// LS Electric XG5000 project: 7k_pwm_20190129_HMI타이밍변경
// PLC NewPLC
// module base 0 slot 0: 입출력 모듈:XBM-DN/DP32H2 (DC 24V입력/TR 출력, 32점)
// module base 0 slot 1: 내장위치결정:XBF-PO02E (오픈컬렉터형, 2축)

PROGRAM 7k_pwm (task: 스캔 프로그램)

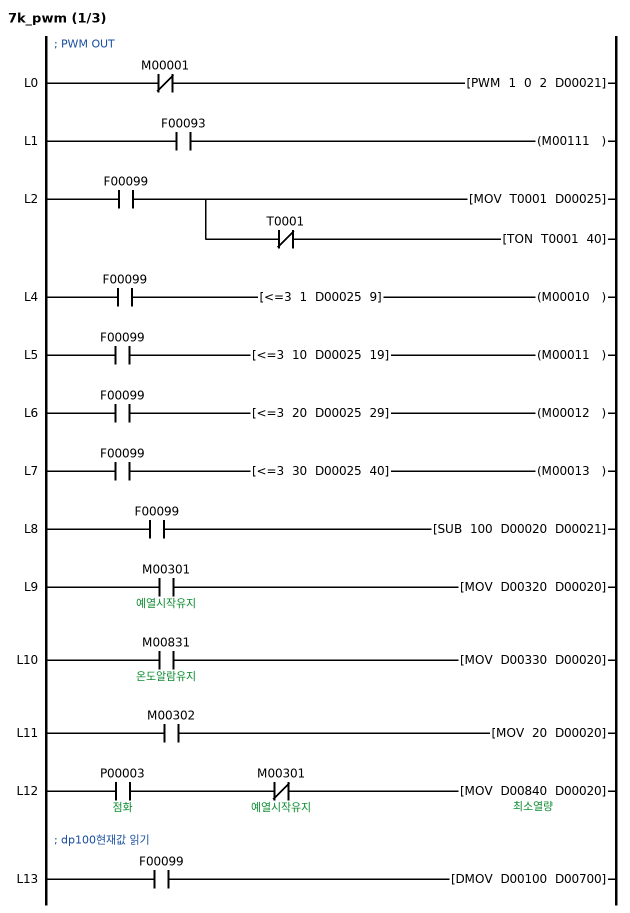
; L0
LOAD NOT  M00001
PWM       1 0 2 D00021
// output comment: PWM OUT
; L1
LOAD      F00093
OUT       M00111
; L2
LOAD      F00099
MOV       T0001 D00025
AND NOT   T0001
TON       T0001 40
; L4
LOAD      F00099
AND<=3    1 D00025 9
OUT       M00010
; L5
LOAD      F00099
AND<=3    10 D00025 19
OUT       M00011
; L6
LOAD      F00099
AND<=3    20 D00025 29
OUT       M00012
; L7
LOAD      F00099
AND<=3    30 D00025 40
OUT       M00013
; L8
LOAD      F00099
SUB       100 D00020 D00021
; L9
LOAD      M00301	// 예열시작유지
MOV       D00320 D00020
; L10
LOAD      M00831	// 온도알람유지
MOV       D00330 D00020
; L11
LOAD      M00302
MOV       20 D00020
; L12
LOAD      P00003	// 점화
AND NOT   M00301	// 예열시작유지
MOV       D00840 D00020	// 최소열량
; L13
LOAD      F00099
DMOV      D00100 D00700
// output comment: dp100현재값 읽기

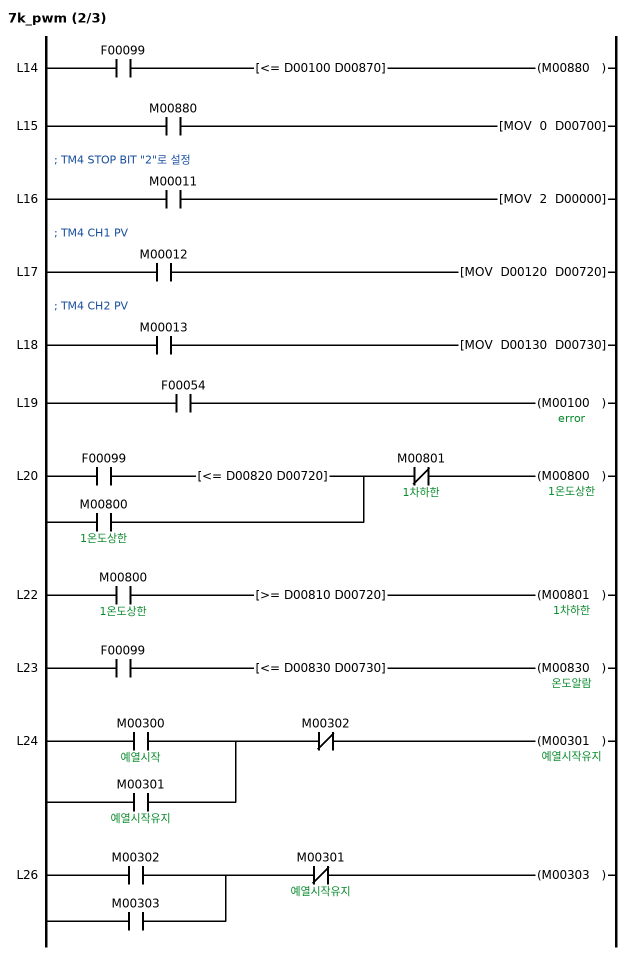
; L14
LOAD      F00099
AND<=     D00100 D00870
OUT       M00880
; L15
LOAD      M00880
MOV       0 D00700
; L16
LOAD      M00011
MOV       2 D00000
// output comment: TM4 STOP BIT "2"로 설정
; L17
LOAD      M00012
MOV       D00120 D00720
// output comment: TM4 CH1 PV
; L18
LOAD      M00013
MOV       D00130 D00730
// output comment: TM4 CH2 PV
; L19
LOAD      F00054
OUT       M00100	// error
; L20
LOAD      F00099
AND<=     D00820 D00720
OR        M00800	// 1온도상한
AND NOT   M00801	// 1차하한
OUT       M00800	// 1온도상한
; L22
LOAD      M00800	// 1온도상한
AND>=     D00810 D00720
OUT       M00801	// 1차하한
; L23
LOAD      F00099
AND<=     D00830 D00730
OUT       M00830	// 온도알람
; L24
LOAD      M00300	// 예열시작
OR        M00301	// 예열시작유지
AND NOT   M00302
OUT       M00301	// 예열시작유지
; L26
LOAD      M00302
OR        M00303
AND NOT   M00301	// 예열시작유지
OUT       M00303

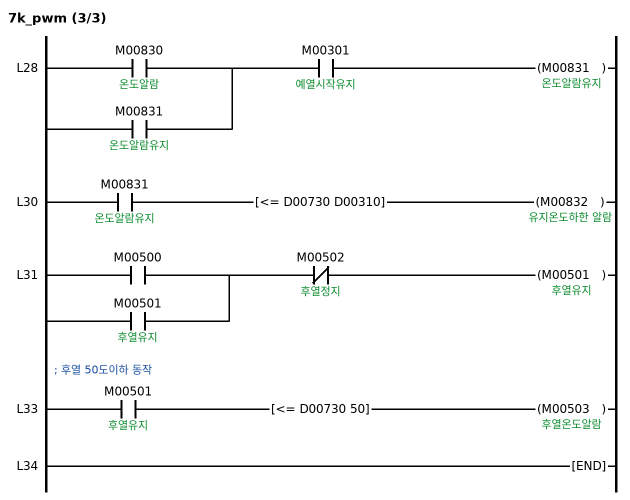
; L28
LOAD      M00830	// 온도알람
OR        M00831	// 온도알람유지
AND       M00301	// 예열시작유지
OUT       M00831	// 온도알람유지
; L30
LOAD      M00831	// 온도알람유지
AND<=     D00730 D00310
OUT       M00832	// 유지온도하한 알람
; L31
LOAD      M00500
OR        M00501	// 후열유지
AND NOT   M00502	// 후열정지
OUT       M00501	// 후열유지
; L33
LOAD      M00501	// 후열유지
AND<=     D00730 50
OUT       M00503	// 후열온도알람
// output comment: 후열 50도이하 동작
; L34
END

PROGRAM 타이머 (task: 스캔 프로그램)

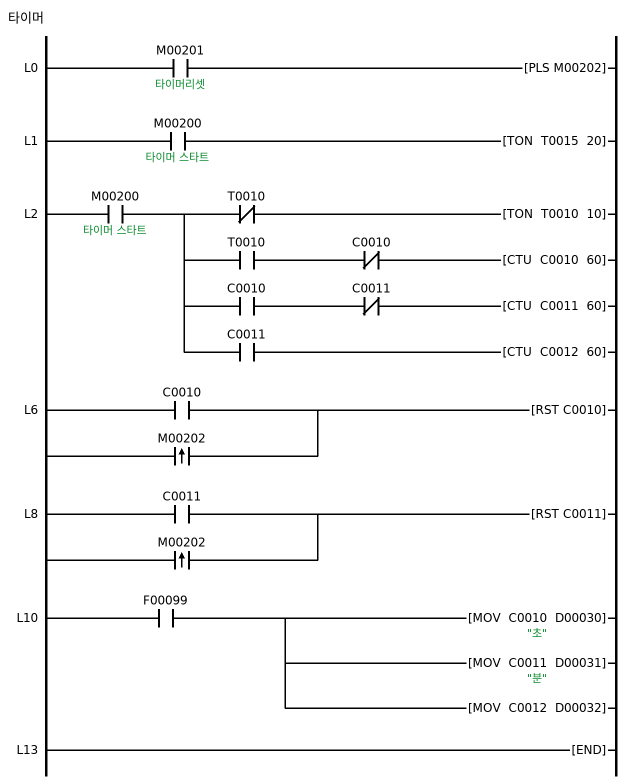
; L0
LOAD      M00201	// 타이머리셋
OUTP      M00202
; L1
LOAD      M00200	// 타이머 스타트
TON       T0015 20
; L2
LOAD      M00200	// 타이머 스타트
MPUSH
AND NOT   T0010
TON       T0010 10
MLOAD
AND       T0010
AND NOT   C0010
CTU       C0010 60
MLOAD
AND       C0010
AND NOT   C0011
CTU       C0011 60
MPOP
AND       C0011
CTU       C0012 60
; L6
LOAD      C0010
ORP       M00202
RST       C0010
; L8
LOAD      C0011
ORP       M00202
RST       C0011
; L10
LOAD      F00099
MOV       C0010 D00030	// "초"
MOV       C0011 D00031	// "분"
MOV       C0012 D00032
; L13
END

PROGRAM control (task: 스캔 프로그램)

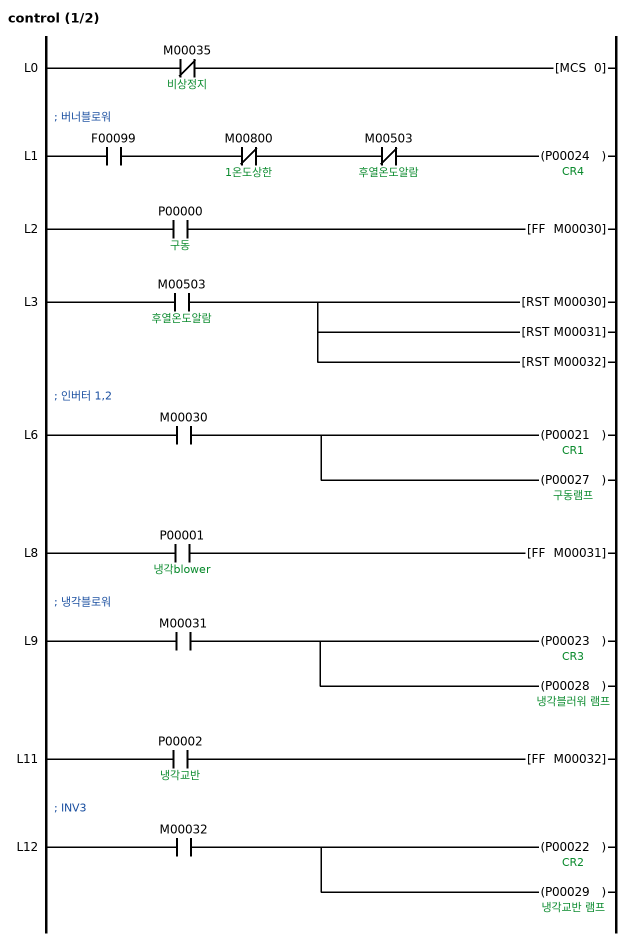
; L0
LOAD NOT  M00035	// 비상정지
MCS       0
; L1
LOAD      F00099
AND NOT   M00800	// 1온도상한
AND NOT   M00503	// 후열온도알람
OUT       P00024	// CR4
// output comment: 버너블로워
; L2
LOAD      P00000	// 구동
FF        M00030
; L3
LOAD      M00503	// 후열온도알람
RST       M00030
RST       M00031
RST       M00032
; L6
LOAD      M00030
OUT       P00021	// CR1
OUT       P00027	// 구동램프
// output comment: 인버터 1,2
; L8
LOAD      P00001	// 냉각blower
FF        M00031
; L9
LOAD      M00031
OUT       P00023	// CR3
OUT       P00028	// 냉각블러워 램프
// output comment: 냉각블로워
; L11
LOAD      P00002	// 냉각교반
FF        M00032
; L12
LOAD      M00032
OUT       P00022	// CR2
OUT       P00029	// 냉각교반 램프
// output comment: INV3

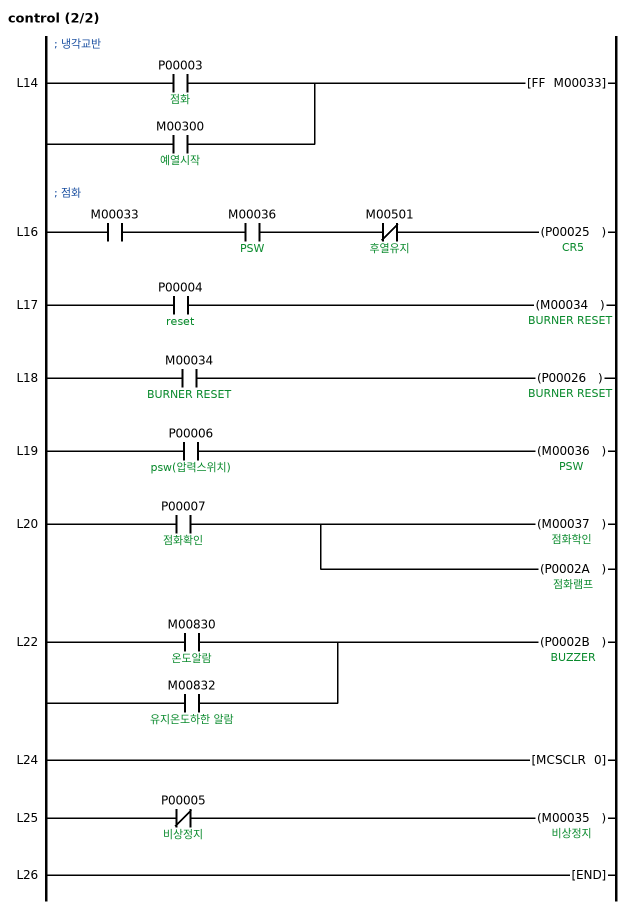
; L14
LOAD      P00003	// 점화
OR        M00300	// 예열시작
FF        M00033
// output comment: 냉각교반
; L16
LOAD      M00033
AND       M00036	// PSW
AND NOT   M00501	// 후열유지
OUT       P00025	// CR5
// output comment: 점화
; L17
LOAD      P00004	// reset
OUT       M00034	// BURNER RESET
; L18
LOAD      M00034	// BURNER RESET
OUT       P00026	// BURNER RESET
; L19
LOAD      P00006	// psw(압력스위치)
OUT       M00036	// PSW
; L20
LOAD      P00007	// 점화확인
OUT       M00037	// 점화학인
OUT       P0002A	// 점화램프
; L22
LOAD      M00830	// 온도알람
OR        M00832	// 유지온도하한 알람
OUT       P0002B	// BUZZER
; L24
MCSCLR    0
; L25
LOAD NOT  P00005	// 비상정지
OUT       M00035	// 비상정지
; L26
END

PROGRAM 10단스위치 (task: 스캔 프로그램)

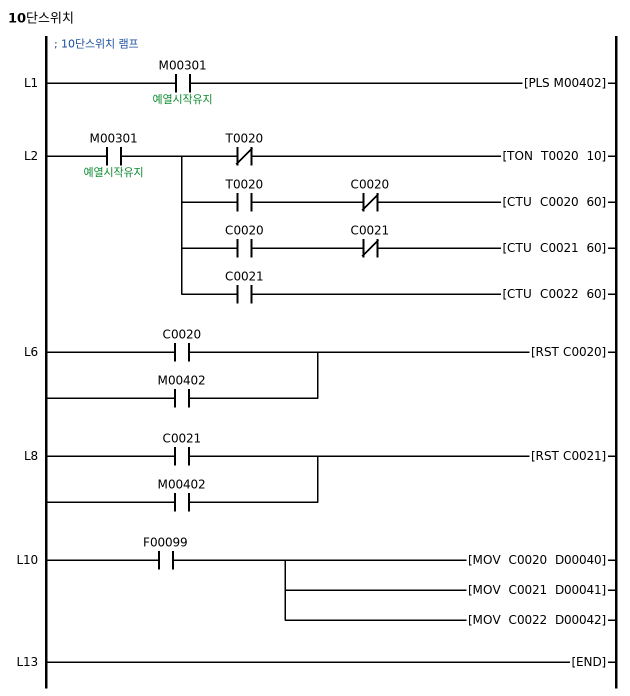
// 10단스위치 램프
; L1
LOAD      M00301	// 예열시작유지
OUTP      M00402
; L2
LOAD      M00301	// 예열시작유지
MPUSH
AND NOT   T0020
TON       T0020 10
MLOAD
AND       T0020
AND NOT   C0020
CTU       C0020 60
MLOAD
AND       C0020
AND NOT   C0021
CTU       C0021 60
MPOP
AND       C0021
CTU       C0022 60
; L6
LOAD      C0020
OR        M00402
RST       C0020
; L8
LOAD      C0021
OR        M00402
RST       C0021
; L10
LOAD      F00099
MOV       C0020 D00040
MOV       C0021 D00041
MOV       C0022 D00042
; L13
END

VARIABLES AND COMMENTS (devices not used above)
P00020	BIT	BURNER PWM
M01001	BIT	0%
M01002	BIT	10%
M01003	BIT	20%
M01004	BIT	30%
M01005	BIT	40%
M01006	BIT	50%
M01007	BIT	60%
M01008	BIT	70%
M01009	BIT	80%
M0100A	BIT	90%
M0100B	BIT	100%
M02001	BIT	0% PL
M02002	BIT	10% PL
M02003	BIT	20% PL
M02004	BIT	30% PL
M02005	BIT	40% PL
M02006	BIT	50% PL
M02007	BIT	60% PL
M02008	BIT	70% PL
M02009	BIT	80% PL
M0200A	BIT	90% PL
M0200B	BIT	100% PL
M03001	BIT	0% PL ON
M03002	BIT	10% PL ON
M03003	BIT	20% PL ON
M03004	BIT	30% PL ON
M03005	BIT	40% PL ON
M03006	BIT	50% PL ON
M03007	BIT	60% PL ON
M03008	BIT	70% PL ON
M03009	BIT	80% PL ON
M0300A	BIT	90% PL ON